// TIA Portal V16 export
VAR_GLOBAL   // PLC tag table "IO Table"
   Send AT %I256 : Bool;   // Tag
END_VAR
